FUNCTION_BLOCK carousel_belt
  (* Standard: 61499-2 *)
  (* Version 0.1, 2015-00-16, Th?o, PC_THEO *)
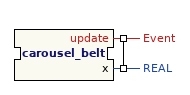
  EVENT_OUTPUT
    update WITH x;
  END_EVENT
  VAR_OUTPUT
    x : REAL;
  END_VAR
  VAR
    beta : REAL;
  END_VAR
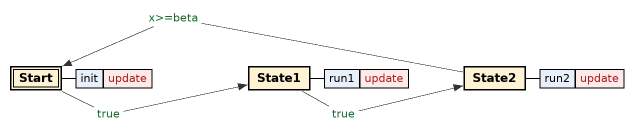
  EC_STATES
    Start : init -> update;
    State1 : run1 -> update;
    State2 : run2 -> update;
  END_STATES
  EC_TRANSITIONS
    Start TO State1 := true;
    State1 TO State2 := true;
    State2 TO Start := x>=beta;
  END_TRANSITIONS
  ALGORITHM init IN C:
me->x=0;
me->beta=10;
  END_ALGORITHM
  ALGORITHM run1 IN C:
//me->x=me->x+1;
me->x=3;
//printf("icecream, %f\n", me->x);
  END_ALGORITHM
  ALGORITHM run2 IN C:
me->x=me->beta;
  END_ALGORITHM
END_FUNCTION_BLOCK
